PROGRAM MAIN
VAR
	nCase 					: INT;
	HwStart 		AT%I* 	: BOOL;
	HwStop  		AT%I* 	: BOOL;
	HwReset 		AT%I* 	: BOOL;
	xOn 			AT%Q* 	: BOOL;
	xRequestReset 	AT%Q* 	: BOOL;
	xError 			AT%Q* 	: BOOL;
		
	VoltageSP 			  	: LREAL := 300;
	rTrigSwitchon 		  	: R_trig;
	fTrigSwitchOff		  	: F_trig;
	Chargtimer 				: ton;
	
	SwitchOn				: BOOL;
	
	TcRestart :TC_Restart;
	Restart : BOOL;
	busy : BOOL;

END_VAR



IF GVL_Safety.HWStart OR hwstart THEN
	GVL_Safety.Run  := TRUE;
	GVL_Safety.Start := TRUE;
END_IF

IF  NOT GVL_Safety.HWStop THEN
	GVL_Safety.Run  := FALSE;
	GVL_Safety.Start := FALSE;
END_IF
		


IF gvl_safety.SaeftyOk THEN
	gvl_safety.HWSafetyOk := TRUE;
ELSE	
	gvl_safety.HWSafetyOk := FALSE;
END_IF

IF NOT gvl_safety.SafetyInRun THEN
	gvl_safety.HWerror := TRUE;
ELSE	
	gvl_safety.HWerror := FALSE;
END_IF

rTrigSwitchon(clk := HwStart );
fTrigSwitchOff(clk:= HwStop );


 Chargtimer(in := SwitchOn ,pt := T#1M, q=>GVL_IO.ChargingResistor);

IF rTrigSwitchon.Q THEN
	GVL_IO.VoltageSet := GVL_IO.VoltageAct;
	SwitchOn := TRUE;
ELSIF fTrigSwitchOff.Q THEN
	SwitchOn := FALSE;
	GVL_IO.VoltageSet :=   0;
END_IF



IF (VoltageSP-2) > GVL_IO.VoltageAct AND  GVL_IO.Voltageset <VoltageSP AND SwitchOn THEN
	GVL_IO.VoltageSet := GVL_IO.VoltageSet +0.1;
END_IF



IF GVL_IO.hwReset OR HwReset THEN
	GVL_IO.ControlDrive1121 := 16#FF;
	GVL_Safety.Reset := TRUE;
	GVL_IO.PowerSupplyReset := TRUE;
ELSE 	
	GVL_IO.ControlDrive1121 := 16#0;
	GVL_Safety.Reset := FALSE;
	GVL_IO.PowerSupplyReset := FALSE;
END_IF


TcRestart(
	NETID:= , 
	RESTART:=Restart , 
	TMOUT:= , 
	BUSY=> , 
	ERR=> , 
	ERRID=> );

END_PROGRAM

(* stored: Version 1.1.0.1, ProductVersion 3.1.4026.8
   POU MAIN: Id {1b4dff48-5fc4-4640-872d-67c650f13b5e}, SpecialFunc None *)
